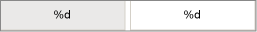
VISUALIZATION VISU_ConfigUINTEntry  // 257x32
VAR_IN_OUT
    active : UINT;
    editable : UINT;
END_VAR
    Textfield (0,0 125x30), "%d", text variable: active, input disabled if: TRUE
    Textfield (130,0 125x30), "%d", text variable: editable, colour toggle: editable <> active
        OnMouseClick: write the text variable via Default
END_VISUALIZATION

(* stored: Version 1.1.0.1, ProductVersion 3.1.0.36
   Visu VISU_ConfigUINTEntry: Id {47f090a5-e2bc-4833-a454-e2d7f84625ee} *)
